% RSLogix 500 project COFFEE_MAKER_BAK001.RSS, saved by version 8.30.00.16 %
PROJECT "UNTITLED"    % processor: Bul.1763 MicroLogix 1100 Series B %

PROGRAM FILES
  LAD 2   13 rungs

DATA FILES
  O0 OUTPUT  4 elements
  I1 INPUT  6 elements
  S2 STATUS  66 elements
  B3 BINARY  1 elements
  T4 TIMER  3 elements
  C5 COUNTER  1 elements
  R6 CONTROL  1 elements
  N7 INTEGER  1 elements
  F8 FLOAT  1 elements

LADDER 2
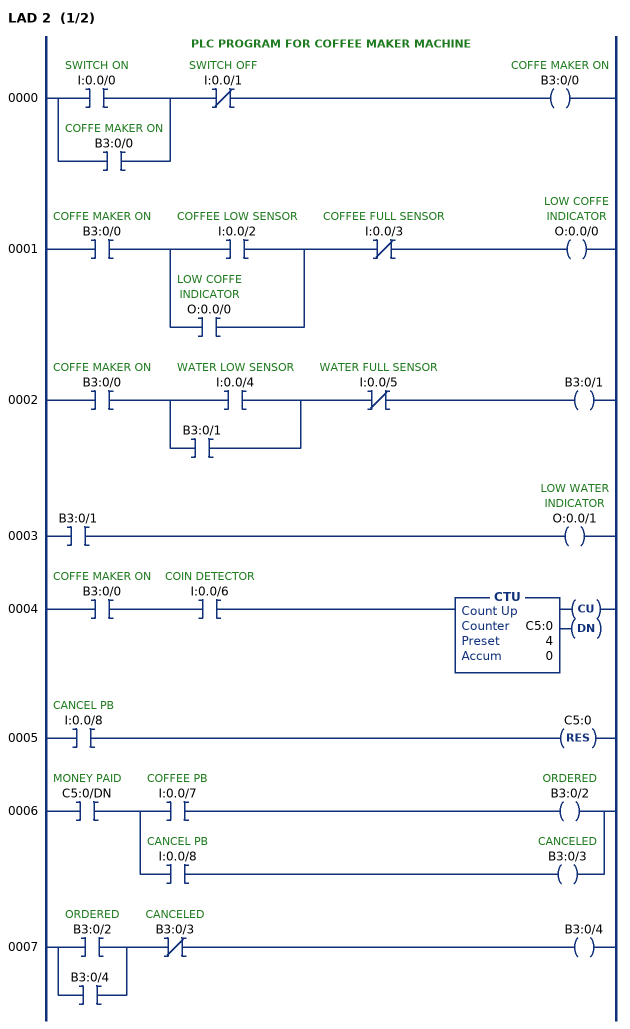
% Rung: 0 %
% TITLE: PLC PROGRAM FOR COFFEE MAKER MACHINE %
SOR BST XIC I:0.0/0 NXB XIC B3:0/0 BND XIO I:0.0/1 OTE B3:0/0 EOR
%   I:0.0/0  "SWITCH ON" %
%   B3:0/0  "COFFE MAKER ON" %
%   I:0.0/1  "SWITCH OFF" %
% Rung: 1 %
SOR XIC B3:0/0 BST XIC I:0.0/2 NXB XIC O:0.0/0 BND XIO I:0.0/3 OTE O:0.0/0 EOR
%   B3:0/0  "COFFE MAKER ON" %
%   I:0.0/2  "COFFEE LOW SENSOR" %
%   O:0.0/0  "LOW COFFE INDICATOR" %
%   I:0.0/3  "COFFEE FULL SENSOR" %
% Rung: 2 %
SOR XIC B3:0/0 BST XIC I:0.0/4 NXB XIC B3:0/1 BND XIO I:0.0/5 OTE B3:0/1 EOR
%   B3:0/0  "COFFE MAKER ON" %
%   I:0.0/4  "WATER LOW SENSOR" %
%   I:0.0/5  "WATER FULL SENSOR" %
% Rung: 3 %
SOR XIC B3:0/1 OTE O:0.0/1 EOR
%   O:0.0/1  "LOW WATER INDICATOR" %
% Rung: 4 %
SOR XIC B3:0/0 XIC I:0.0/6 CTU C5:0 4 0 EOR
%   B3:0/0  "COFFE MAKER ON" %
%   I:0.0/6  "COIN DETECTOR" %
% Rung: 5 %
SOR XIC I:0.0/8 RES C5:0 EOR
%   I:0.0/8  "CANCEL PB" %
% Rung: 6 %
SOR XIC C5:0/DN BST XIC I:0.0/7 OTE B3:0/2 NXB XIC I:0.0/8 OTE B3:0/3 BND EOR
%   C5:0/DN  "MONEY PAID" %
%   I:0.0/7  "COFFEE PB" %
%   B3:0/2  "ORDERED" %
%   I:0.0/8  "CANCEL PB" %
%   B3:0/3  "CANCELED" %
% Rung: 7 %
SOR BST XIC B3:0/2 NXB XIC B3:0/4 BND XIO B3:0/3 OTE B3:0/4 EOR
%   B3:0/2  "ORDERED" %
%   B3:0/3  "CANCELED" %

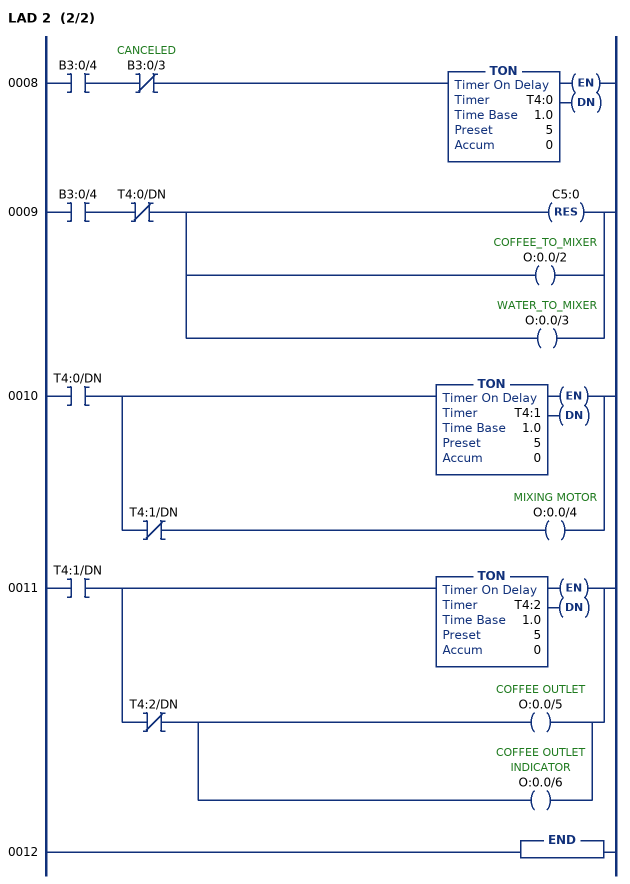
% Rung: 8 %
SOR XIC B3:0/4 XIO B3:0/3 TON T4:0 1.0 5 0 EOR
%   B3:0/3  "CANCELED" %
% Rung: 9 %
SOR XIC B3:0/4 XIO T4:0/DN BST RES C5:0 NXB OTE O:0.0/2 NXB OTE O:0.0/3 BND EOR
%   O:0.0/2  "COFFEE_TO_MIXER" %
%   O:0.0/3  "WATER_TO_MIXER" %
% Rung: 10 %
SOR XIC T4:0/DN BST TON T4:1 1.0 5 0 NXB XIO T4:1/DN OTE O:0.0/4 BND EOR
%   O:0.0/4  "MIXING MOTOR" %
% Rung: 11 %
SOR XIC T4:1/DN BST TON T4:2 1.0 5 0 NXB XIO T4:2/DN BST OTE O:0.0/5 NXB OTE O:0.0/6 BND BND EOR
%   O:0.0/5  "COFFEE OUTLET" %
%   O:0.0/6  "COFFEE OUTLET INDICATOR" %
% Rung: 12 %
SOR END EOR

DATA TABLE (non-zero values as saved)
DATA T4
% .PRE .ACC %
% T4:0 % 5 0
% T4:1 % 5 0
% T4:2 % 5 0
DATA C5
% .PRE .ACC %
% C5:0 % 4 0
